# EPICS autosave request: iocBoot/sioc-emit2-im01/sioc-emit2-im01.req
file "lcls2toro.req" AREA=EMIT2,POS=170
